{attribute 'GeneratedUsingTerminal: EJ2918-0000-0017'}
{attribute addProperty BoxType "EJ2918-0000-0017"}
{attribute addProperty Id "FSOEAT %Q*FSOE_2DC96D3115"}
{attribute addProperty CRC "768645799"}
{attribute addProperty Size "15"}
TYPE FSoE_Outputs_2DD09AA7 EXTENDS OutputBase_10CEE7DE :
STRUCT
	{attribute addProperty Name "FSOE"}
	FSOE AT %Q* : FSOE_2DC96D31;
END_STRUCT
END_TYPE
